PROGRAM MAIN
VAR
END_VAR

END_PROGRAM

(* stored: Version 1.1.0.1
   POU MAIN: Id {e4f67c36-33b2-4f37-bbe8-f91e24f68352} *)
